FUNCTION_BLOCK Bohrmaschine IMPLEMENTS I_Machine
VAR
	ipLogger: I_MachineLogger;
	bohrer: Bohrkopf;
	axesManager: AxesManager;

	// Zustand der Maschine
	eZustand: E_MACHINE_STATES := E_MACHINE_STATES.eWaiting;

	// anzufahrende Punkte
	aPunkte: ARRAY [0..3] OF ST_2DPoint;
	nCurIdx: USINT := 0;
	
	// Hilfsvariablen Visualisierung
	nProgressStep: USINT := 0;

	bRunning: BOOL := FALSE;
	stHomePoint: ST_2DPoint := (x := 0, y := 0);
END_VAR


axesManager();
bohrer();

CASE eZustand OF
	E_MACHINE_STATES.eWaiting:
		// idle

	E_MACHINE_STATES.eStopping:
		Stopping();

	E_MACHINE_STATES.eMoving:
		Moving();

	E_MACHINE_STATES.eDrilling:
		Drilling();
END_CASE

METHOD PRIVATE Config : BOOL
VAR
	rBreite: LREAL;
	rLaenge: LREAL;
END_VAR
VAR CONSTANT
	// Abstand des Bohrlochs zur Aussenseite
	// TODO später als Input
	rAbstand: LREAL := 10;
END_VAR
// die vier Koordinaten berechnen und speichern, TODO später: Bohrlochtiefe + Abstand

rBreite := GVL_Config.stConfig.rBreite;
rLaenge := GVL_Config.stConfig.rLaenge;

// Punkt 1
aPunkte[0].x := rAbstand;
aPunkte[0].y := rAbstand;

// Punkt 2
aPunkte[1].x := 10;
aPunkte[1].y := rBreite - rAbstand;

// Punkt 3
aPunkte[2].x := rLaenge - rAbstand;
aPunkte[2].y := rBreite - rAbstand;

// Punkt 4
aPunkte[3].x := rLaenge - rAbstand;
aPunkte[3].y := rAbstand;
END_METHOD

METHOD PRIVATE Drill : BOOL
eZustand := E_MACHINE_STATES.eDrilling;
END_METHOD

METHOD PRIVATE Drilling : BOOL
VAR_INPUT
END_VAR
VAR
	bGebohrt: BOOL := FALSE;
END_VAR
// Bohren
bohrer.Bohren(bDone => bGebohrt);
IF(bGebohrt) THEN
	// Progressbar + 1
	GVL_Control.nProgress := GVL_Control.nProgress + 1;
	ipLogger.LogBohrung(axesManager.CurrentPoint);

	MoveNext();
END_IF
END_METHOD

METHOD FB_init : BOOL
VAR_INPUT
	bInitRetains : BOOL; // if TRUE, the retain variables are initialized (warm start / cold start)
	bInCopyCode : BOOL;  // if TRUE, the instance afterwards gets moved into the copy code (online change)
	ipLogger: I_MachineLogger;
END_VAR
THIS^.ipLogger := ipLogger;
END_METHOD

METHOD PRIVATE MoveNext : BOOL
// Nächsten Anfahrtspunkt setzen. Bohrloch oder Home.

// Wenn alle Bohrlöcher abgefahren wurden -> go Home / stop
IF nCurIdx > 3 THEN
	Stop();
ELSE // nächsten Bohrpunkt setzen
	axesManager.Start(aPunkte[nCurIdx]);
	nCurIdx := nCurIdx + 1;	
	eZustand := E_MACHINE_STATES.eMoving;
END_IF
END_METHOD

METHOD PRIVATE Moving : BOOL
VAR_INPUT
END_VAR

IF axesManager.bPunktAngefahren THEN
	F_Log('Moved To:');
	axesManager.LogAxes();
	axesManager.Stop();
	// Progressbar + 1
	GVL_Control.nProgress := GVL_Control.nProgress + 1;
	
	ipLogger.LogPunktAngefahren(axesManager.CurrentPoint);
	// Achsenbewegungen abgeschlossen, Drill
	Drill();
END_IF
END_METHOD

METHOD PUBLIC Start : BOOL
THIS^.bRunning := TRUE;
GVL_Control.bIsRunning := TRUE;
// Progressbar = 0
GVL_Control.nProgress := 0;
Config();
axesManager.Enable(bEnableAxes := TRUE);
MoveNext();
ipLogger.LogStart();
END_METHOD

METHOD PUBLIC Stop : BOOL
// wenn intern durch Ende gestoppt wurde, benötigt es keinen Stop von aussen
IF THIS^.bRunning = FALSE THEN
	RETURN;
END_IF

THIS^.bRunning := FALSE;
GVL_Control.bRun := FALSE;
axesManager.Stop();
bohrer.Stop();
eZustand := E_MACHINE_STATES.eStopping;
nCurIdx := 0;
END_METHOD

METHOD PRIVATE Stopping : BOOL
VAR
	bBohrerStopped: BOOL := FALSE;
END_VAR
// Warten bis der Bohrkopf oben ist, dann zum Nullpunkt fahren
bohrer.Stopping(bDone => bBohrerStopped);
IF bBohrerStopped THEN
	F_Log('Fahre Home');
	axesManager.Start(stHomePoint);
END_IF

IF axesManager.bPunktAngefahren THEN
	F_Log('Home:');
	axesManager.LogAxes();
	axesManager.Stop();
	eZustand := E_MACHINE_STATES.eWaiting;
	GVL_Control.bIsRunning := FALSE;
	// Progressbar + 1
	GVL_Control.nProgress := 9;
	ipLogger.LogStop();
END_IF
END_METHOD

END_FUNCTION_BLOCK

(* stored: Version 1.1.0.1, ProductVersion 3.1.4024.3
   POU Bohrmaschine: Id {9e061517-3285-4418-b8f4-b3a23dd6952d}, SpecialFunc None
   Method Config: Id {25dde089-95eb-4734-88fc-9c38d9b5ac13}
   Method Drill: Id {f6a05a08-ae6b-4538-9167-85cc33480e82}
   Method Drilling: Id {de0fd246-a5eb-4e47-9ece-8ff9cbdbcce5}
   Method FB_init: Id {11913734-036a-4115-89b4-2a8ed7163773}
   Method MoveNext: Id {cd40f332-95bc-4193-ac41-7e2ebbe98ced}
   Method Moving: Id {62a2e616-9837-49bd-a407-f2e14bff6ecb}
   Method Start: Id {77e5359d-b759-40cf-a154-1c37eaa6ebbf}
   Method Stop: Id {c65ecb49-f392-471e-8cd2-32ba1727ca52}
   Method Stopping: Id {70e2eab1-d929-470f-b1c1-4867fe667962} *)
